// SIMATIC S7-200 project (STEP 7-Micro/WIN), CPU 224XP REL 02.00

SYMBOL_TABLE USER1
scadrx           VD23
encdrx           VW10
motorx           Q0.0
hdencodrix       VD10
scada_t_zad      M4.1
scadrxvod        M5.1
scada_start      M3.1
scada_time       VD100
scada_svd        M7.1
scada_vd         VD110
motorz           Q0.1
END_SYMBOL_TABLE

ORGANIZATION_BLOCK Fast_Encoder_Simple_S:OB1
TITLE=S7-200 + Fast Encoder + Simple-Scada
// v1.0
// 
// #NVJOB Nicholas Veselov (independent developer) - https://nvjob.pro, http://nvjob.dx.am
// 
BEGIN
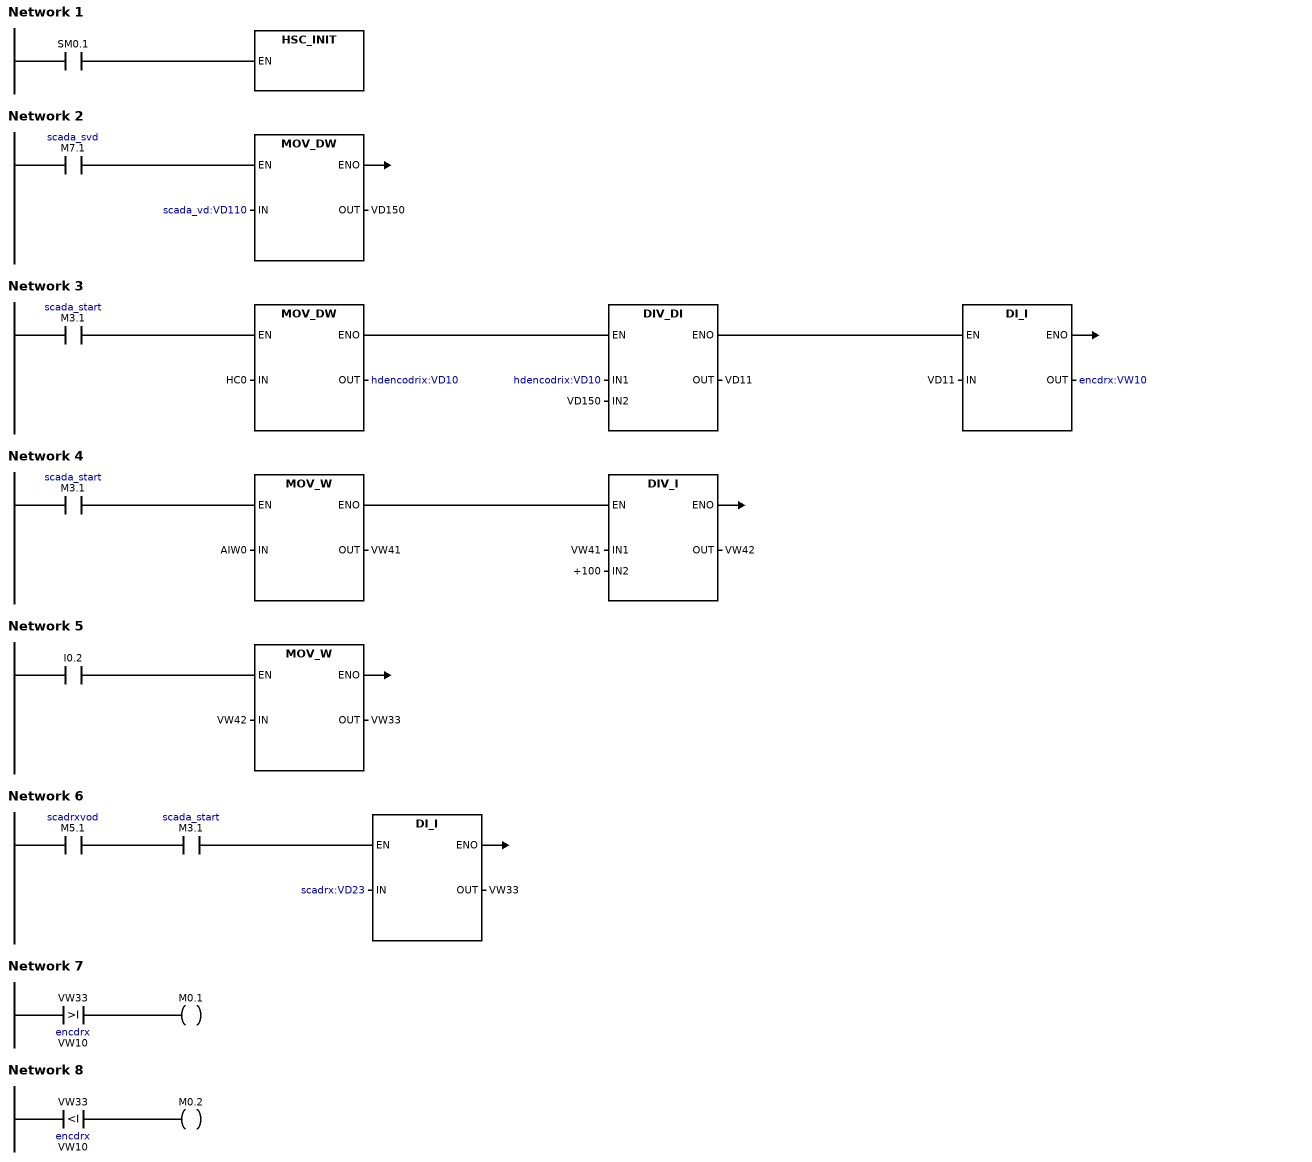
Network 1
LD     SM0.1
CALL   HSC_INIT:SBR1
Network 2
LD     scada_svd:M7.1
MOVD   scada_vd:VD110, VD150
Network 3
LD     scada_start:M3.1
MOVD   HC0, hdencodrix:VD10
AENO
MOVD   hdencodrix:VD10, VD11
AENO
/D     VD150, VD11
AENO
DTI    VD11, encdrx:VW10
Network 4
LD     scada_start:M3.1
MOVW   AIW0, VW41
AENO
MOVW   VW41, VW42
/I     +100, VW42
Network 5
LD     I0.2
MOVW   VW42, VW33
Network 6
LD     scadrxvod:M5.1
A      scada_start:M3.1
DTI    scadrx:VD23, VW33
Network 7
LDW>   VW33, encdrx:VW10
=      M0.1
Network 8
LDW<   VW33, encdrx:VW10
=      M0.2
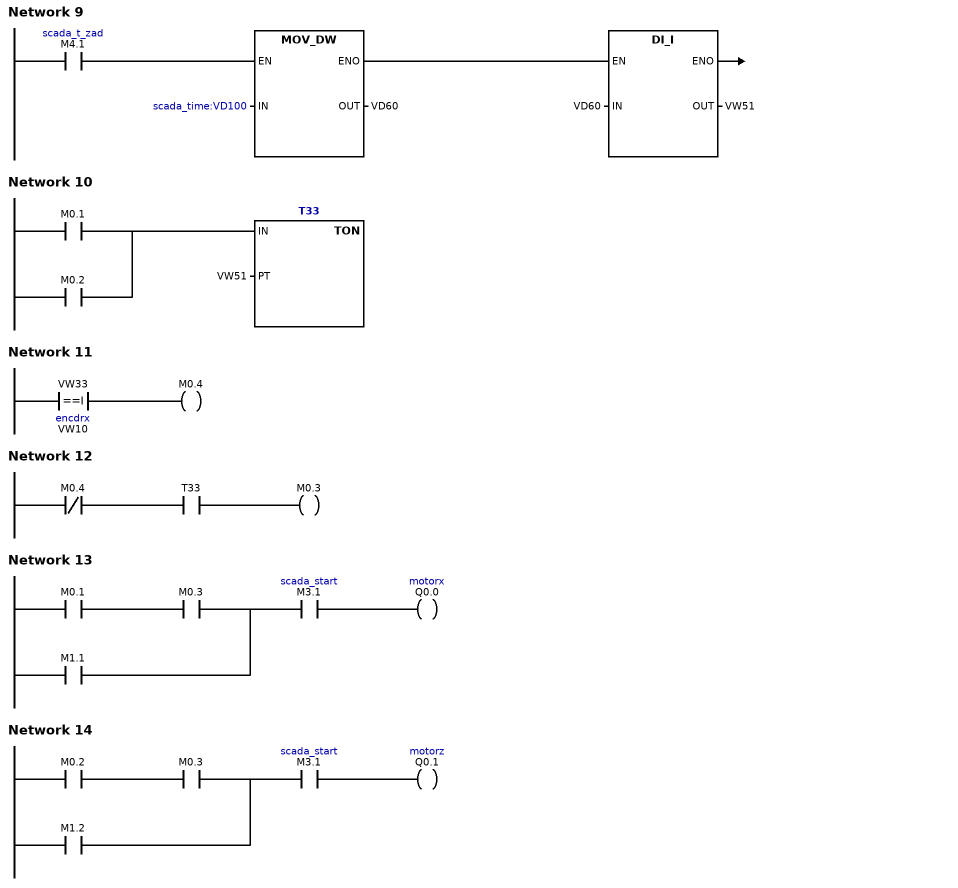
Network 9
LD     scada_t_zad:M4.1
MOVD   scada_time:VD100, VD60
AENO
DTI    VD60, VW51
Network 10
LD     M0.1
O      M0.2
TON    T33, VW51
Network 11
LDW=   VW33, encdrx:VW10
=      M0.4
Network 12
LDN    M0.4
A      T33
=      M0.3
Network 13
LD     M0.1
A      M0.3
O      M1.1
A      scada_start:M3.1
=      motorx:Q0.0
Network 14
LD     M0.2
A      M0.3
O      M1.2
A      scada_start:M3.1
=      motorz:Q0.1
END_ORGANIZATION_BLOCK

SUBROUTINE_BLOCK HSC_INIT:SBR1
TITLE=
BEGIN
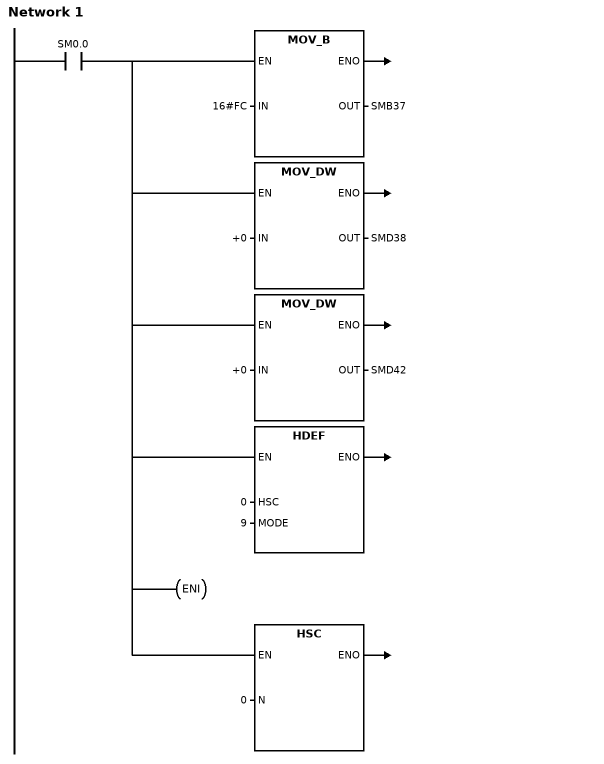
Network 1
LD     SM0.0
MOVB   16#FC, SMB37
MOVD   +0, SMD38
MOVD   +0, SMD42
HDEF   0, 9
ENI
HSC    0
END_SUBROUTINE_BLOCK
